{attribute 'call_after_init'}
FUNCTION_BLOCK FB_LeakMonitor_Test EXTENDS FB_TestSuite
VAR_INPUT
END_VAR
VAR_OUTPUT
END_VAR
VAR
END_VAR

LOTAOTriggers1();
LOTAOTriggers2();
LOTAOLatches();
LOTAOResets();
LOTNLTriggers1();
LOTNLTriggers2();
LOTNLLatches();
LOTNLResets();
LOCOTriggers1();
LOCOTriggers2();
LOCOLatches();
LOCOResets();
LUTTriggers1();
LUTTriggers2();
LUTLatches();
LUTResets();
LIRTriggers1();
LIRTriggers2();
LIRLatches();
LIRResets();
NoLeak();

METHOD LIRLatches
VAR
	fbLeakMonitor : FB_LeakMonitor;
	stLeakBoundaries : ST_LeakBoundaries;
END_VAR
TEST('LeakInsideRacksLatches');

fbLeakMonitor := F_LeakMonitor_LIR_1(stBoundaries => stLeakBoundaries);

// Leak Error should stay latched even when inputs go back to normal
fbLeakMonitor(
	bLeakDetected := FALSE,
	stBound := stLeakBoundaries
);

AssertTrue(fbLeakMonitor.bLeakInsideRacks, 'Leak error did not stay latched');

TEST_FINISHED();
END_METHOD

METHOD LIRResets
VAR
	fbLeakMonitor : FB_LeakMonitor;
	stLeakBoundaries : ST_LeakBoundaries;
END_VAR
TEST('LeakInsideRacksResets');

fbLeakMonitor := F_LeakMonitor_LIR_1(stBoundaries => stLeakBoundaries);

// Error should be resettable
fbLeakMonitor.Reset();
fbLeakMonitor(bLeakDetected := FALSE, stBound := stLeakBoundaries);
AssertFalse(fbLeakMonitor.bLeakInsideRacks, 'Leak error did not reset');

TEST_FINISHED();
END_METHOD

METHOD LIRTriggers1
VAR
	fbLeakMonitor : FB_LeakMonitor := F_LeakMonitor_LIR_1();
END_VAR
TEST('LeakInsideRacksTriggers1');

AssertTrue(fbLeakMonitor.bLeakInsideRacks, 'Leak error did not trigger');

TEST_FINISHED();
END_METHOD

METHOD LIRTriggers2
VAR
	fbLeakMonitor : FB_LeakMonitor := F_LeakMonitor_LIR_2();
END_VAR
TEST('LeakInsideRacksTriggers2');

AssertTrue(fbLeakMonitor.bLeakInsideRacks, 'Leak error did not trigger');

TEST_FINISHED();
END_METHOD

METHOD LOCOLatches
VAR
	fbLeakMonitor : FB_LeakMonitor;
	stLeakBoundaries : ST_LeakBoundaries;
END_VAR
TEST('LeakOpcpaCarbideOnLatches');

fbLeakMonitor := F_LeakMonitor_LOCO_1(stBoundaries => stLeakBoundaries);

// Leak Error should stay latched even when inputs go back to normal
fbLeakMonitor(
	bLeakDetected := FALSE,
	stBound := stLeakBoundaries,
);
AssertTrue(fbLeakMonitor.bLeakOpcpaCarbideOn, 'Leak error did not stay latched');

TEST_FINISHED();
END_METHOD

METHOD LOCOResets
VAR
	fbLeakMonitor : FB_LeakMonitor;
	stLeakBoundaries : ST_LeakBoundaries;
END_VAR
TEST('LeakOpcpaCarbideOnResets');

fbLeakMonitor := F_LeakMonitor_LOCO_1(stBoundaries => stLeakBoundaries);

// Error should be resettable
fbLeakMonitor.Reset();
fbLeakMonitor(bLeakDetected := FALSE, stBound := stLeakBoundaries);
AssertFalse(fbLeakMonitor.bLeakOpcpaCarbideOn, 'Leak error did not reset');

TEST_FINISHED();
END_METHOD

METHOD LOCOTriggers1
VAR
	fbLeakMonitor : FB_LeakMonitor := F_LeakMonitor_LOCO_1();
END_VAR
TEST('LeakOpcpaCarbideOnTriggers11');

AssertTrue(fbLeakMonitor.bLeakOpcpaCarbideOn, 'Leak error did not trigger');

TEST_FINISHED();
END_METHOD

METHOD LOCOTriggers2
VAR
	fbLeakMonitor : FB_LeakMonitor := F_LeakMonitor_LOCO_2();
END_VAR
TEST('LeakOpcpaCarbideOnTriggers2');

AssertTrue(fbLeakMonitor.bLeakOpcpaCarbideOn, 'Leak error did not trigger');

TEST_FINISHED();
END_METHOD

METHOD LOTAOLatches
VAR
	fbLeakMonitor : FB_LeakMonitor;
	stLeakBoundaries : ST_LeakBoundaries;
END_VAR
TEST('LeakOpticalTableAmphosOnLatches');

fbLeakMonitor := F_LeakMonitor_LOTAO_1(stBoundaries => stLeakBoundaries);

// Leak Error should stay latched even when inputs go back to normal
fbLeakMonitor(
	bLeakDetected := FALSE,
	stBound := stLeakBoundaries
);

AssertTrue(fbLeakMonitor.bLeakOpticalTableAmphosOn, 'Leak error did not stay latched');

TEST_FINISHED();
END_METHOD

METHOD LOTAOResets
VAR
	fbLeakMonitor : FB_LeakMonitor;
	stLeakBoundaries : ST_LeakBoundaries;
END_VAR
TEST('LeakOpticalTableAmphosOnResets');

fbLeakMonitor := F_LeakMonitor_LOTAO_1(stBoundaries => stLeakBoundaries);

// Error should be resettable
fbLeakMonitor.Reset();
fbLeakMonitor(bLeakDetected := FALSE, stBound := stLeakBoundaries);
AssertFalse(fbLeakMonitor.bLeakOpticalTableAmphosOn, 'Leak error did not reset');

TEST_FINISHED();
END_METHOD

METHOD LOTAOTriggers1
VAR
	fbLeakMonitor : FB_LeakMonitor := F_LeakMonitor_LOTAO_1();
END_VAR
TEST('LeakOpticalTableAmphosOnTriggers1');

AssertTrue(fbLeakMonitor.bLeakOpticalTableAmphosOn, 'Leak error did not trigger');

TEST_FINISHED();
END_METHOD

METHOD LOTAOTriggers2
VAR
	fbLeakMonitor : FB_LeakMonitor := F_LeakMonitor_LOTAO_2();
END_VAR
TEST('LeakOpticalTableAmphosOnTriggers2');

AssertTrue(fbLeakMonitor.bLeakOpticalTableAmphosOn, 'Leak error did not trigger');

TEST_FINISHED();
END_METHOD

METHOD LOTNLLatches
VAR
	fbLeakMonitor : FB_LeakMonitor;
	stLeakBoundaries : ST_LeakBoundaries;
END_VAR
TEST('LeakOpticalTableNoLaserLatches');

fbLeakMonitor := F_LeakMonitor_LOTNL_1(stBoundaries => stLeakBoundaries);

// Leak Error should stay latched even when inputs go back to normal
fbLeakMonitor(
	bLeakDetected := FALSE,
	stBound := stLeakBoundaries
);
AssertTrue(fbLeakMonitor.bLeakOpticalTableNoLaser, 'Leak error did not stay latched');

TEST_FINISHED();
END_METHOD

METHOD LOTNLResets
VAR
	fbLeakMonitor : FB_LeakMonitor;
	stLeakBoundaries : ST_LeakBoundaries;
END_VAR
TEST('LeakOpticalTableNoLaserResets');

fbLeakMonitor := F_LeakMonitor_LOTNL_1(stBoundaries => stLeakBoundaries);

// Error should be resettable
fbLeakMonitor.Reset();
fbLeakMonitor(bLeakDetected := FALSE, stBound := stLeakBoundaries);
AssertFalse(fbLeakMonitor.bLeakOpticalTableNoLaser, 'Leak error did not reset');

TEST_FINISHED();
END_METHOD

METHOD LOTNLTriggers1
VAR
	fbLeakMonitor : FB_LeakMonitor := F_LeakMonitor_LOTNL_1();
END_VAR
TEST('LeakOpticalTableNoLaserTriggers1');

AssertTrue(fbLeakMonitor.bLeakOpticalTableNoLaser, 'Leak error did not trigger');

TEST_FINISHED();
END_METHOD

METHOD LOTNLTriggers2
VAR
	fbLeakMonitor : FB_LeakMonitor := F_LeakMonitor_LOTNL_2();
END_VAR
TEST('LeakOpticalTableNoLaserTriggers2');

AssertTrue(fbLeakMonitor.bLeakOpticalTableNoLaser, 'Leak error did not trigger');

TEST_FINISHED();
END_METHOD

METHOD LUTLatches
VAR
	fbLeakMonitor : FB_LeakMonitor;
	stLeakBoundaries : ST_LeakBoundaries;
END_VAR
TEST('LeakUnderTableLatches');

fbLeakMonitor := F_LeakMonitor_LUT_1(stBoundaries => stLeakBoundaries);

// Leak Error should stay latched even when inputs go back to normal
fbLeakMonitor(
	bLeakDetected := FALSE,
	stBound := stLeakBoundaries,
);
AssertTrue(fbLeakMonitor.bLeakUnderTable, 'Leak error did not stay latched');

TEST_FINISHED();
END_METHOD

METHOD LUTResets
VAR
	fbLeakMonitor : FB_LeakMonitor;
	stLeakBoundaries : ST_LeakBoundaries;
END_VAR
TEST('LeakUnderTableResets');

fbLeakMonitor := F_LeakMonitor_LUT_1(stBoundaries => stLeakBoundaries);

// Error should be resettable
fbLeakMonitor.Reset();
fbLeakMonitor(bLeakDetected := FALSE, stBound := stLeakBoundaries);
AssertFalse(fbLeakMonitor.bLeakUnderTable, 'Leak error did not reset');

TEST_FINISHED();
END_METHOD

METHOD LUTTriggers1
VAR
	fbLeakMonitor : FB_LeakMonitor := F_LeakMonitor_LUT_1();
END_VAR
TEST('LeakUnderTableTriggers1');

AssertTrue(fbLeakMonitor.bLeakUnderTable, 'Leak error did not trigger');

TEST_FINISHED();
END_METHOD

METHOD LUTTriggers2
VAR
	fbLeakMonitor : FB_LeakMonitor := F_LeakMonitor_LUT_2();
END_VAR
TEST('LeakUnderTableTriggers2');

AssertTrue(fbLeakMonitor.bLeakUnderTable, 'Leak error did not trigger');

TEST_FINISHED();
END_METHOD

METHOD NoLeak
VAR
	fbLeakMonitor : FB_LeakMonitor;
	stLeakBoundaries : ST_LeakBoundaries := F_LeakBoundaries();
END_VAR
TEST('NoLeak');

fbLeakMonitor(
	bLeakDetected := FALSE,
	bAmphosOn := TRUE,
	bCarbideOn := TRUE,
	stBound := stLeakBoundaries,
	nLocationResistance := stLeakBoundaries.nLMax6,
);
AssertFalse(fbLeakMonitor.bLeakOpticalTableAmphosOn OR fbLeakMonitor.bLeakOpticalTableNoLaser OR fbLeakMonitor.bLeakOpcpaCarbideOn OR fbLeakMonitor.bLeakUnderTable
	OR fbLeakMonitor.bLeakInsideRacks, 'Leak fasely detected');
	
TEST_FINISHED();
END_METHOD

END_FUNCTION_BLOCK

(* stored: Version 1.1.0.1, ProductVersion 3.1.4024.0
   POU FB_LeakMonitor_Test: Id {e7e4db1c-c6e4-470e-83ff-3b26cb0a2d29}, SpecialFunc None
   Method LIRLatches: Id {7fa63837-983e-4ea3-b140-cc5e94a25d71}
   Method LIRResets: Id {8803dd34-02cd-4ab8-966e-a8464ebce051}
   Method LIRTriggers1: Id {4fb51dcb-69a6-416e-babc-44de1e243bf1}
   Method LIRTriggers2: Id {3d9f057f-9248-4e2e-9721-76c0e985ceaa}
   Method LOCOLatches: Id {43be45d4-0016-4d8c-9274-e2c7b6562fad}
   Method LOCOResets: Id {9be9b98f-b5d8-4350-a5d4-724d6e93fb88}
   Method LOCOTriggers1: Id {095ea75a-a116-46d9-8b51-781b925f9570}
   Method LOCOTriggers2: Id {5e1b77b1-e349-423c-9e8d-f9c58c7f5794}
   Method LOTAOLatches: Id {469a5268-7865-4459-bd89-a6f020c4ffee}
   Method LOTAOResets: Id {ec9fa339-8ada-417c-bdbe-c033a3b02bbd}
   Method LOTAOTriggers1: Id {275d5fe8-71c1-4e3b-94ed-a98f9ca832ad}
   Method LOTAOTriggers2: Id {0a483ae8-0dd5-4013-bc2a-37ae27b2ac2d}
   Method LOTNLLatches: Id {0be33797-17ae-4571-9257-62fb45685960}
   Method LOTNLResets: Id {585568e5-9bb8-4000-ad33-7b3f12cdd84e}
   Method LOTNLTriggers1: Id {e5a3d21a-9a36-455b-82b8-42ef73a8ca61}
   Method LOTNLTriggers2: Id {1c0de105-19e9-40f2-96a4-a1341bb6140c}
   Method LUTLatches: Id {aeb67bed-623e-4b3b-9088-6d04b93d352d}
   Method LUTResets: Id {7b9715cc-9225-499c-96ab-b2b68564ea25}
   Method LUTTriggers1: Id {04d682b9-6af2-49ee-8b34-e73b4822969c}
   Method LUTTriggers2: Id {f6e258a6-9cc0-45eb-8bec-ef7098c23dd1}
   Method NoLeak: Id {5c679667-707c-40bf-9b54-79b1bd0e59be} *)
